// TIA Portal V18 program export: 1 tag tables, 0 data types, 0 data blocks, 7 code blocks (in call order from the OBs), 1 instance data blocks

VAR_GLOBAL   // PLC tag table "Default tag table"
   Tag_1 AT %M0.0 : Bool;
   Tag_2 AT %M1.0 : Bool;
END_VAR

ORGANIZATION_BLOCK "Main"   // OB1, LAD, ProgramCycle
TITLE = "Main Program Sweep (Cycle)"
{ S7_Optimized_Access := 'TRUE' }
VERSION : 0.1
// stored: AutoNumber true, IsIECCheckEnabled false, SetENOAutomatically false
   VAR_INPUT
      Initial_Call : Bool;   // Initial call of this OB
      Remanence : Bool;   // =True, if remanent data are available
   END_VAR
BEGIN

REGION Network 1
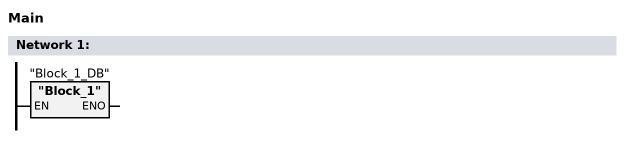
   RUNG wire#powerrail
      "Block_1_DB"()
   END_RUNG
   // the same network as SCL:
   "Block_1_DB"();   // "Block_1"
END_REGION
END_ORGANIZATION_BLOCK

FUNCTION_BLOCK "Block_1"
{ S7_Optimized_Access := 'TRUE' }
VERSION : 0.1

BEGIN
	IF "Tag_1" = 1 THEN
	    "Tag_2" := 1;
	END_IF;
	
END_FUNCTION_BLOCK

FUNCTION "Block_LADDER" : Void   // FC5, LAD
{ S7_Optimized_Access := 'TRUE' }
VERSION : 0.1
// stored: AutoNumber true, IsIECCheckEnabled false, SetENOAutomatically false, UDAEnableTagReadback false
BEGIN

REGION Network 1
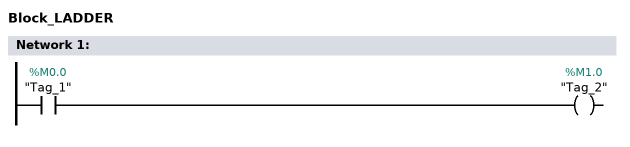
   RUNG wire#powerrail
      Contact( "Tag_1" )
      Coil( "Tag_2" )
   END_RUNG
   // the same network as SCL:
   "Tag_2" := "Tag_1";
END_REGION
END_FUNCTION

FUNCTION "Block_2" : Void
{ S7_Optimized_Access := 'TRUE' }
VERSION : 0.1

BEGIN
	// test block
END_FUNCTION

FUNCTION "Block_3" : Void
{ S7_Optimized_Access := 'TRUE' }
VERSION : 0.1

BEGIN
	// branch test
END_FUNCTION

FUNCTION "Block_4" : Void
{ S7_Optimized_Access := 'TRUE' }
VERSION : 0.1

BEGIN
END_FUNCTION

FUNCTION "Block_5" : Void
{ S7_Optimized_Access := 'TRUE' }
VERSION : 0.1

BEGIN
END_FUNCTION

DATA_BLOCK "Block_1_DB"   // DB1
VERSION : 0.1
// stored: AutoNumber true, InstanceOfName Block_1, InstanceOfType FB
"Block_1"
BEGIN
END_DATA_BLOCK
